FUNCTION_BLOCK Q_StringValue_AIS (* Command Change String Value ( Part 6 - F.24 ) *)
  (* Standard: ISO 11783-6; Description: Copyright (c) 2026 HR Agrartechnik GmbH This program and the accompanying materials are made available under the terms of the Eclipse Public License 2.0 which is available at https://www.eclipse.org/legal/epl-2.0/ SPDX-License-Identifier: EPL-2.0 *)
  (* Version 1.0, 2026-04-13, Franz Höpfinger, HR Agrartechnik GmbH *)
  PACKAGE isobus::UT::Q;
  IMPORT isobus::UT::Q::const::IDs::ID_NULL;
  (* Documentation:
  Command change string value ( Part 6 - F.24 )
   This command is used to change the value of an object. It applies only to objects that have a string value attribute. This FB is an AIS adapter wrapper around Q_StringValue — the same object-type validity rules and the F.24 variable data length / transport protocol behaviour apply.
   Valid Object IDs
   u16ObjId is valid if it falls within one of the following ISO 11783-6 ID ranges (see Q_StringValue, Annex F.24):
    - InputStringField: 8000 – 8999
   - OutputStringField: 11000 – 11999
   - StringVariable: 22000 – 22999
   - InputAttributesObject: 26000 – 26999
    ID_NULL (65535) is not a command target but can be used in INIT to deactivate the FB. Any ID outside these ranges is invalid for commanding.
  *)
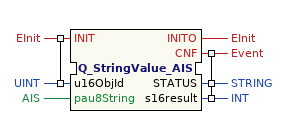
  EVENT_INPUT
    INIT : EInit WITH u16ObjId; (* Service Initialization *)
  END_EVENT
  EVENT_OUTPUT
    INITO : EInit; (* Initialization Confirm *)
    CNF WITH STATUS, s16result; (* Confirmation of Requested Service *)
  END_EVENT
  VAR_INPUT
    u16ObjId : UINT := ID_NULL; (* Object ID *)
  END_VAR
  VAR_OUTPUT
    STATUS : STRING; (* Service Status *)
    s16result : INT; (* retval see description *)
  END_VAR
  SOCKETS
    pau8String : adapter::types::unidirectional::AIS; (* New string value *)
  END_SOCKETS
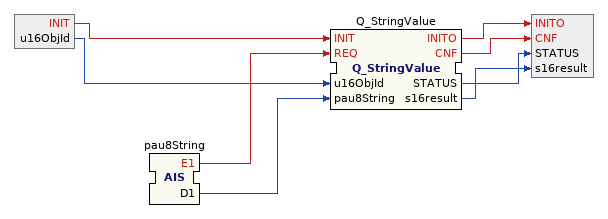
  FBS
    Q_StringValue : isobus::UT::Q::Q_StringValue;
  END_FBS
  EVENT_CONNECTIONS
    INIT TO Q_StringValue.INIT;
    Q_StringValue.INITO TO INITO;
    Q_StringValue.CNF TO CNF;
    pau8String.E1 TO Q_StringValue.REQ;
  END_CONNECTIONS
  DATA_CONNECTIONS
    u16ObjId TO Q_StringValue.u16ObjId;
    pau8String.D1 TO Q_StringValue.pau8String;
    Q_StringValue.STATUS TO STATUS;
    Q_StringValue.s16result TO s16result;
  END_CONNECTIONS
END_FUNCTION_BLOCK
